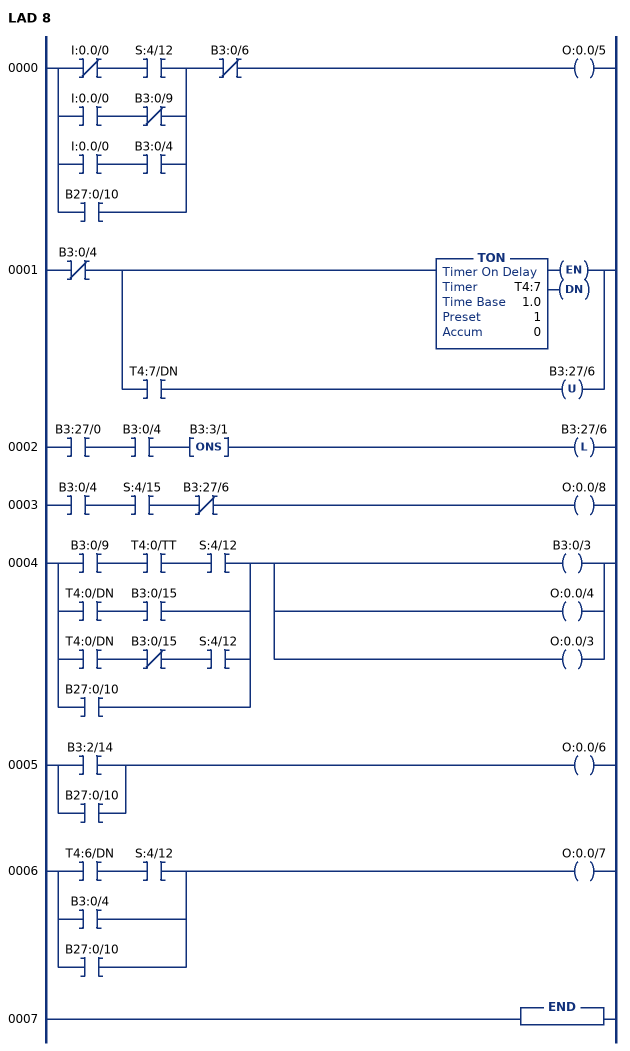
% Rung: 0 %
SOR BST XIO I:0.0/0 XIC S:4/12 NXB XIC I:0.0/0 XIO B3:0/9 NXB XIC I:0.0/0 XIC B3:0/4 NXB XIC B27:0/10 BND XIO B3:0/6 OTE O:0.0/5 EOR
% Rung: 1 %
SOR XIO B3:0/4 BST TON T4:7 1.0 1 0 NXB XIC T4:7/DN OTU B3:27/6 BND EOR
% Rung: 2 %
SOR XIC B3:27/0 XIC B3:0/4 ONS B3:3/1 OTL B3:27/6 EOR
% Rung: 3 %
SOR XIC B3:0/4 XIC S:4/15 XIO B3:27/6 OTE O:0.0/8 EOR
% Rung: 4 %
SOR BST XIC B3:0/9 XIC T4:0/TT XIC S:4/12 NXB XIC T4:0/DN XIC B3:0/15 NXB XIC T4:0/DN XIO B3:0/15 XIC S:4/12 NXB XIC B27:0/10 BND BST OTE B3:0/3 NXB OTE O:0.0/4 NXB OTE O:0.0/3 BND EOR
% Rung: 5 %
SOR BST XIC B3:2/14 NXB XIC B27:0/10 BND OTE O:0.0/6 EOR
% Rung: 6 %
SOR BST XIC T4:6/DN XIC S:4/12 NXB XIC B3:0/4 NXB XIC B27:0/10 BND OTE O:0.0/7 EOR
% Rung: 7 %
SOR END EOR

LADDER 9
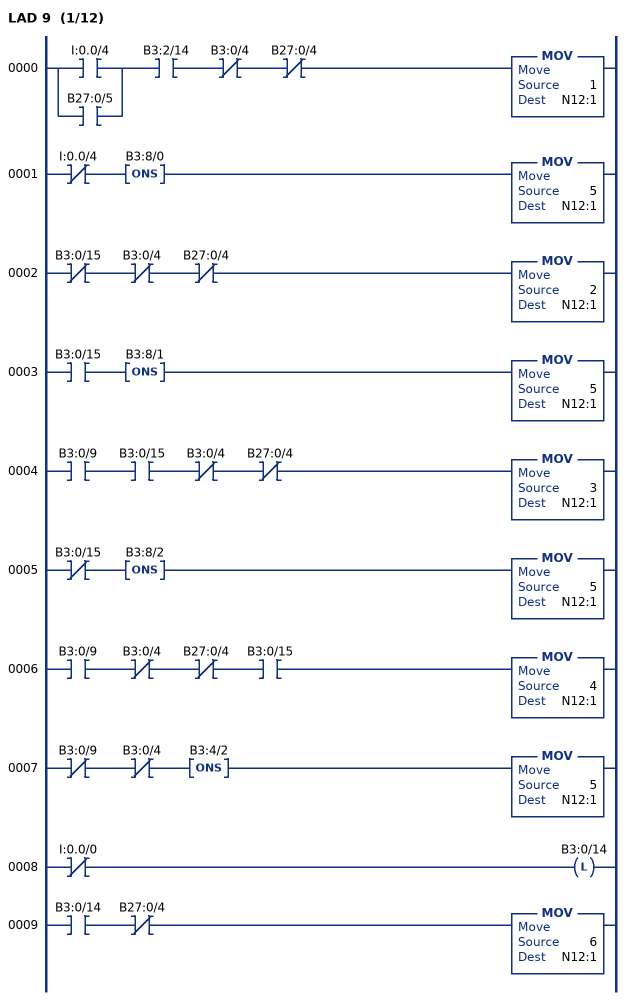
% Rung: 0 %
SOR BST XIC I:0.0/4 NXB XIC B27:0/5 BND XIC B3:2/14 XIO B3:0/4 XIO B27:0/4 MOV 1 N12:1 EOR
% Rung: 1 %
SOR XIO I:0.0/4 ONS B3:8/0 MOV 5 N12:1 EOR
% Rung: 2 %
SOR XIO B3:0/15 XIO B3:0/4 XIO B27:0/4 MOV 2 N12:1 EOR
% Rung: 3 %
SOR XIC B3:0/15 ONS B3:8/1 MOV 5 N12:1 EOR
% Rung: 4 %
SOR XIC B3:0/9 XIC B3:0/15 XIO B3:0/4 XIO B27:0/4 MOV 3 N12:1 EOR
% Rung: 5 %
SOR XIO B3:0/15 ONS B3:8/2 MOV 5 N12:1 EOR
% Rung: 6 %
SOR XIC B3:0/9 XIO B3:0/4 XIO B27:0/4 XIC B3:0/15 MOV 4 N12:1 EOR
% Rung: 7 %
SOR XIO B3:0/9 XIO B3:0/4 ONS B3:4/2 MOV 5 N12:1 EOR
% Rung: 8 %
SOR XIO I:0.0/0 OTL B3:0/14 EOR
% Rung: 9 %
SOR XIC B3:0/14 XIO B27:0/4 MOV 6 N12:1 EOR

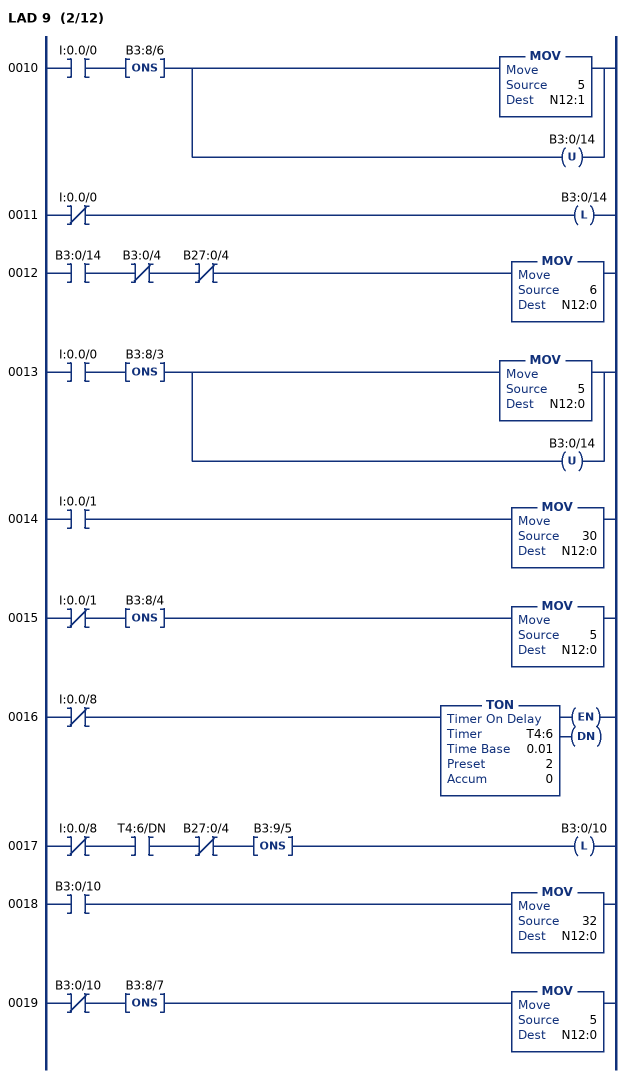
% Rung: 10 %
SOR XIC I:0.0/0 ONS B3:8/6 BST MOV 5 N12:1 NXB OTU B3:0/14 BND EOR
% Rung: 11 %
SOR XIO I:0.0/0 OTL B3:0/14 EOR
% Rung: 12 %
SOR XIC B3:0/14 XIO B3:0/4 XIO B27:0/4 MOV 6 N12:0 EOR
% Rung: 13 %
SOR XIC I:0.0/0 ONS B3:8/3 BST MOV 5 N12:0 NXB OTU B3:0/14 BND EOR
% Rung: 14 %
SOR XIC I:0.0/1 MOV 30 N12:0 EOR
% Rung: 15 %
SOR XIO I:0.0/1 ONS B3:8/4 MOV 5 N12:0 EOR
% Rung: 16 %
SOR XIO I:0.0/8 TON T4:6 0.01 2 0 EOR
% Rung: 17 %
SOR XIO I:0.0/8 XIC T4:6/DN XIO B27:0/4 ONS B3:9/5 OTL B3:0/10 EOR
% Rung: 18 %
SOR XIC B3:0/10 MOV 32 N12:0 EOR
% Rung: 19 %
SOR XIO B3:0/10 ONS B3:8/7 MOV 5 N12:0 EOR

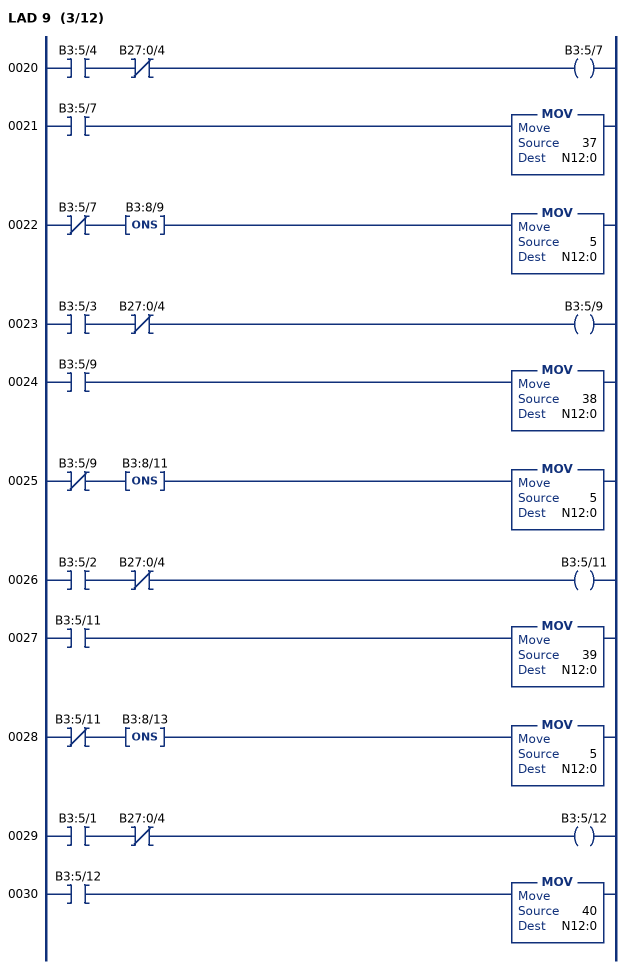
% Rung: 20 %
SOR XIC B3:5/4 XIO B27:0/4 OTE B3:5/7 EOR
% Rung: 21 %
SOR XIC B3:5/7 MOV 37 N12:0 EOR
% Rung: 22 %
SOR XIO B3:5/7 ONS B3:8/9 MOV 5 N12:0 EOR
% Rung: 23 %
SOR XIC B3:5/3 XIO B27:0/4 OTE B3:5/9 EOR
% Rung: 24 %
SOR XIC B3:5/9 MOV 38 N12:0 EOR
% Rung: 25 %
SOR XIO B3:5/9 ONS B3:8/11 MOV 5 N12:0 EOR
% Rung: 26 %
SOR XIC B3:5/2 XIO B27:0/4 OTE B3:5/11 EOR
% Rung: 27 %
SOR XIC B3:5/11 MOV 39 N12:0 EOR
% Rung: 28 %
SOR XIO B3:5/11 ONS B3:8/13 MOV 5 N12:0 EOR
% Rung: 29 %
SOR XIC B3:5/1 XIO B27:0/4 OTE B3:5/12 EOR
% Rung: 30 %
SOR XIC B3:5/12 MOV 40 N12:0 EOR

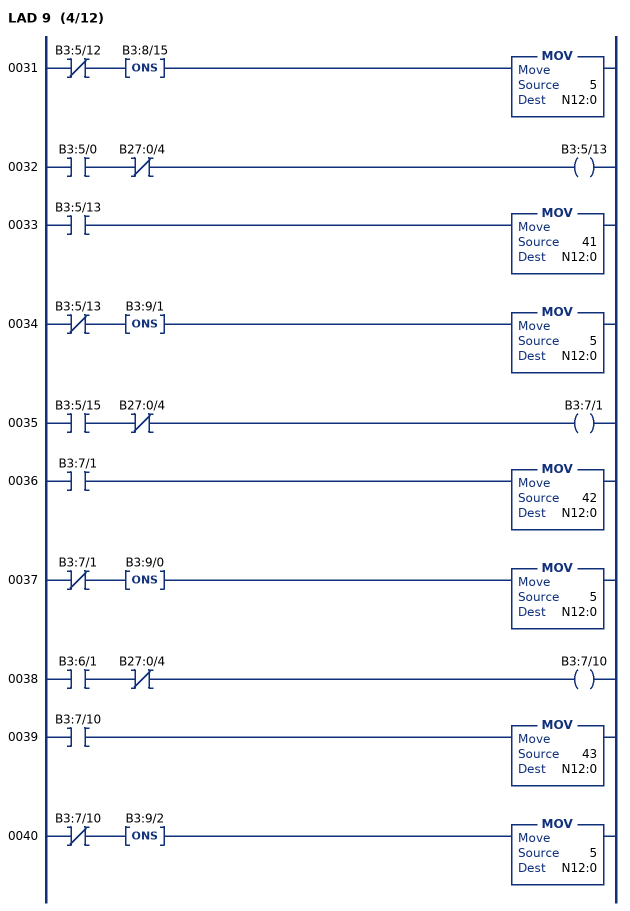
% Rung: 31 %
SOR XIO B3:5/12 ONS B3:8/15 MOV 5 N12:0 EOR
% Rung: 32 %
SOR XIC B3:5/0 XIO B27:0/4 OTE B3:5/13 EOR
% Rung: 33 %
SOR XIC B3:5/13 MOV 41 N12:0 EOR
% Rung: 34 %
SOR XIO B3:5/13 ONS B3:9/1 MOV 5 N12:0 EOR
% Rung: 35 %
SOR XIC B3:5/15 XIO B27:0/4 OTE B3:7/1 EOR
% Rung: 36 %
SOR XIC B3:7/1 MOV 42 N12:0 EOR
% Rung: 37 %
SOR XIO B3:7/1 ONS B3:9/0 MOV 5 N12:0 EOR
% Rung: 38 %
SOR XIC B3:6/1 XIO B27:0/4 OTE B3:7/10 EOR
% Rung: 39 %
SOR XIC B3:7/10 MOV 43 N12:0 EOR
% Rung: 40 %
SOR XIO B3:7/10 ONS B3:9/2 MOV 5 N12:0 EOR

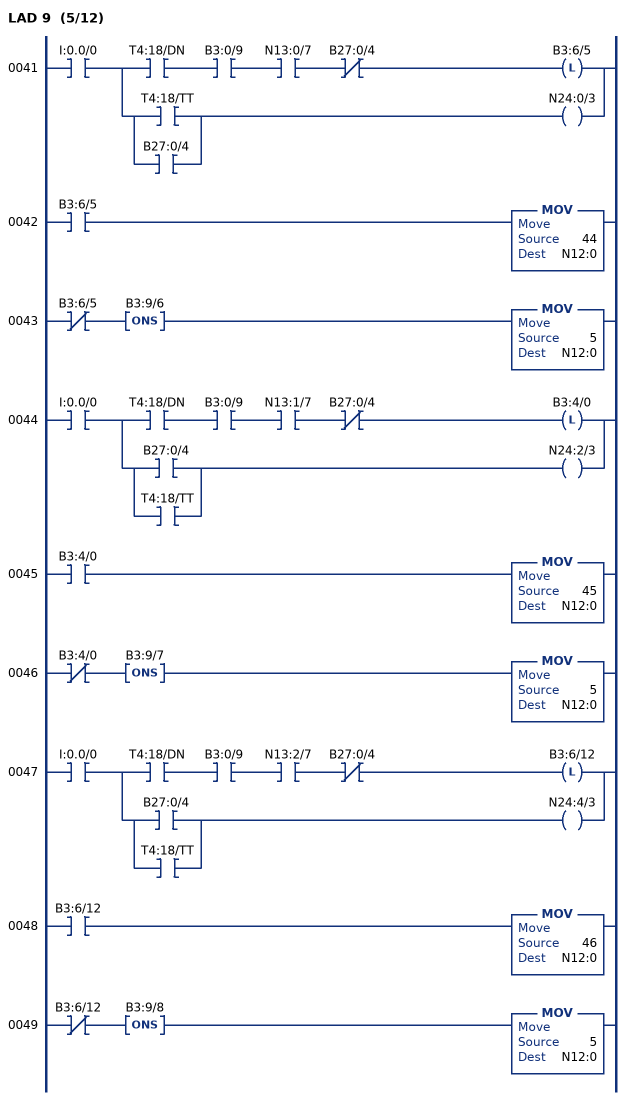
% Rung: 41 %
SOR XIC I:0.0/0 BST XIC T4:18/DN XIC B3:0/9 XIC N13:0/7 XIO B27:0/4 OTL B3:6/5 NXB BST XIC T4:18/TT NXB XIC B27:0/4 BND OTE N24:0/3 BND EOR
% Rung: 42 %
SOR XIC B3:6/5 MOV 44 N12:0 EOR
% Rung: 43 %
SOR XIO B3:6/5 ONS B3:9/6 MOV 5 N12:0 EOR
% Rung: 44 %
SOR XIC I:0.0/0 BST XIC T4:18/DN XIC B3:0/9 XIC N13:1/7 XIO B27:0/4 OTL B3:4/0 NXB BST XIC B27:0/4 NXB XIC T4:18/TT BND OTE N24:2/3 BND EOR
% Rung: 45 %
SOR XIC B3:4/0 MOV 45 N12:0 EOR
% Rung: 46 %
SOR XIO B3:4/0 ONS B3:9/7 MOV 5 N12:0 EOR
% Rung: 47 %
SOR XIC I:0.0/0 BST XIC T4:18/DN XIC B3:0/9 XIC N13:2/7 XIO B27:0/4 OTL B3:6/12 NXB BST XIC B27:0/4 NXB XIC T4:18/TT BND OTE N24:4/3 BND EOR
% Rung: 48 %
SOR XIC B3:6/12 MOV 46 N12:0 EOR
% Rung: 49 %
SOR XIO B3:6/12 ONS B3:9/8 MOV 5 N12:0 EOR

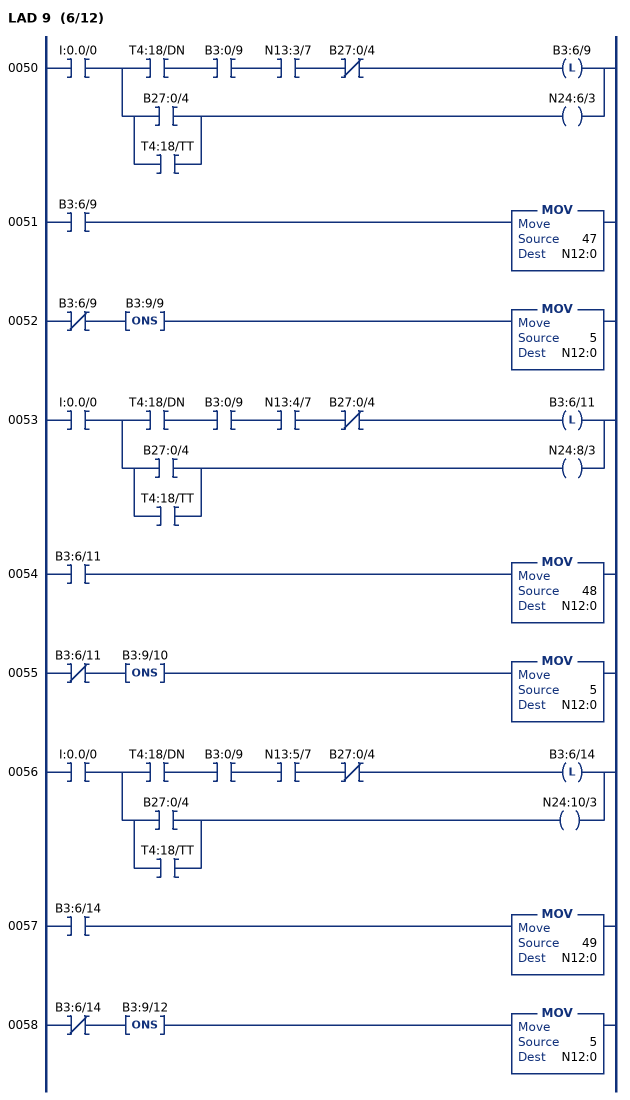
% Rung: 50 %
SOR XIC I:0.0/0 BST XIC T4:18/DN XIC B3:0/9 XIC N13:3/7 XIO B27:0/4 OTL B3:6/9 NXB BST XIC B27:0/4 NXB XIC T4:18/TT BND OTE N24:6/3 BND EOR
% Rung: 51 %
SOR XIC B3:6/9 MOV 47 N12:0 EOR
% Rung: 52 %
SOR XIO B3:6/9 ONS B3:9/9 MOV 5 N12:0 EOR
% Rung: 53 %
SOR XIC I:0.0/0 BST XIC T4:18/DN XIC B3:0/9 XIC N13:4/7 XIO B27:0/4 OTL B3:6/11 NXB BST XIC B27:0/4 NXB XIC T4:18/TT BND OTE N24:8/3 BND EOR
% Rung: 54 %
SOR XIC B3:6/11 MOV 48 N12:0 EOR
% Rung: 55 %
SOR XIO B3:6/11 ONS B3:9/10 MOV 5 N12:0 EOR
% Rung: 56 %
SOR XIC I:0.0/0 BST XIC T4:18/DN XIC B3:0/9 XIC N13:5/7 XIO B27:0/4 OTL B3:6/14 NXB BST XIC B27:0/4 NXB XIC T4:18/TT BND OTE N24:10/3 BND EOR
% Rung: 57 %
SOR XIC B3:6/14 MOV 49 N12:0 EOR
% Rung: 58 %
SOR XIO B3:6/14 ONS B3:9/12 MOV 5 N12:0 EOR

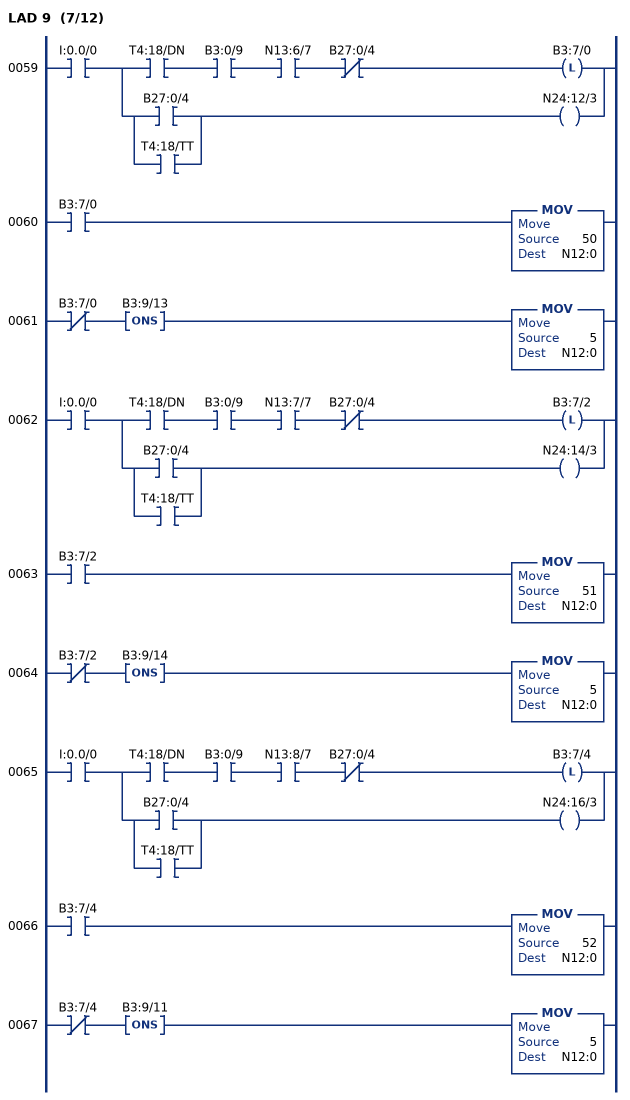
% Rung: 59 %
SOR XIC I:0.0/0 BST XIC T4:18/DN XIC B3:0/9 XIC N13:6/7 XIO B27:0/4 OTL B3:7/0 NXB BST XIC B27:0/4 NXB XIC T4:18/TT BND OTE N24:12/3 BND EOR
% Rung: 60 %
SOR XIC B3:7/0 MOV 50 N12:0 EOR
% Rung: 61 %
SOR XIO B3:7/0 ONS B3:9/13 MOV 5 N12:0 EOR
% Rung: 62 %
SOR XIC I:0.0/0 BST XIC T4:18/DN XIC B3:0/9 XIC N13:7/7 XIO B27:0/4 OTL B3:7/2 NXB BST XIC B27:0/4 NXB XIC T4:18/TT BND OTE N24:14/3 BND EOR
% Rung: 63 %
SOR XIC B3:7/2 MOV 51 N12:0 EOR
% Rung: 64 %
SOR XIO B3:7/2 ONS B3:9/14 MOV 5 N12:0 EOR
% Rung: 65 %
SOR XIC I:0.0/0 BST XIC T4:18/DN XIC B3:0/9 XIC N13:8/7 XIO B27:0/4 OTL B3:7/4 NXB BST XIC B27:0/4 NXB XIC T4:18/TT BND OTE N24:16/3 BND EOR
% Rung: 66 %
SOR XIC B3:7/4 MOV 52 N12:0 EOR
% Rung: 67 %
SOR XIO B3:7/4 ONS B3:9/11 MOV 5 N12:0 EOR

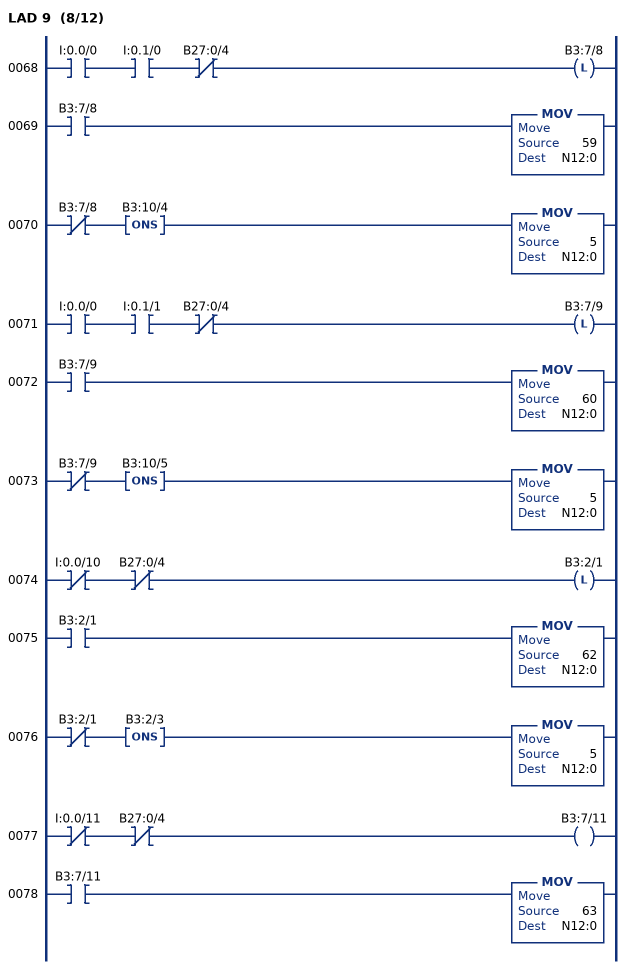
% Rung: 68 %
SOR XIC I:0.0/0 XIC I:0.1/0 XIO B27:0/4 OTL B3:7/8 EOR
% Rung: 69 %
SOR XIC B3:7/8 MOV 59 N12:0 EOR
% Rung: 70 %
SOR XIO B3:7/8 ONS B3:10/4 MOV 5 N12:0 EOR
% Rung: 71 %
SOR XIC I:0.0/0 XIC I:0.1/1 XIO B27:0/4 OTL B3:7/9 EOR
% Rung: 72 %
SOR XIC B3:7/9 MOV 60 N12:0 EOR
% Rung: 73 %
SOR XIO B3:7/9 ONS B3:10/5 MOV 5 N12:0 EOR
% Rung: 74 %
SOR XIO I:0.0/10 XIO B27:0/4 OTL B3:2/1 EOR
% Rung: 75 %
SOR XIC B3:2/1 MOV 62 N12:0 EOR
% Rung: 76 %
SOR XIO B3:2/1 ONS B3:2/3 MOV 5 N12:0 EOR
% Rung: 77 %
SOR XIO I:0.0/11 XIO B27:0/4 OTE B3:7/11 EOR
% Rung: 78 %
SOR XIC B3:7/11 MOV 63 N12:0 EOR

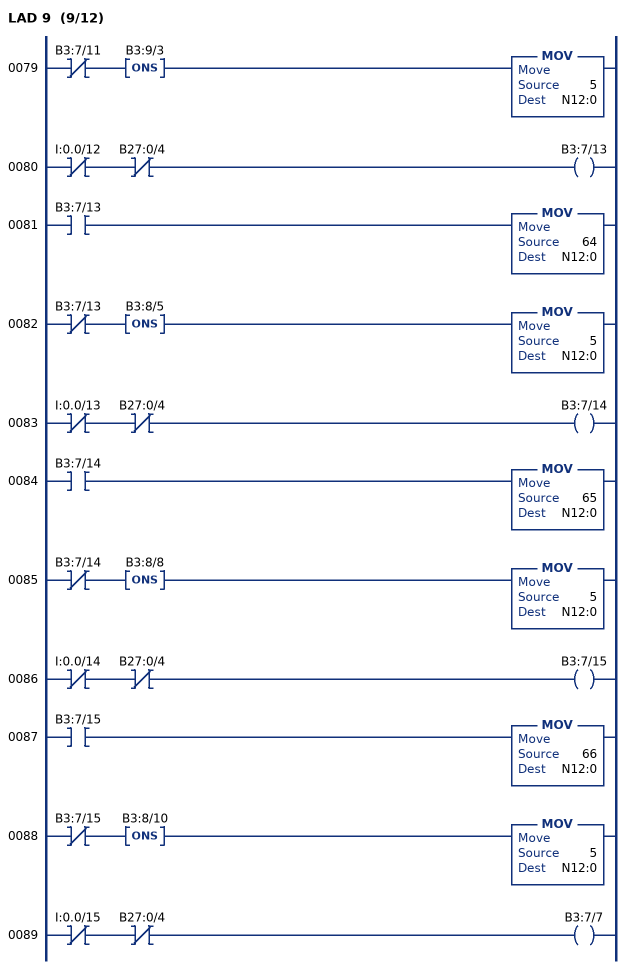
% Rung: 79 %
SOR XIO B3:7/11 ONS B3:9/3 MOV 5 N12:0 EOR
% Rung: 80 %
SOR XIO I:0.0/12 XIO B27:0/4 OTE B3:7/13 EOR
% Rung: 81 %
SOR XIC B3:7/13 MOV 64 N12:0 EOR
% Rung: 82 %
SOR XIO B3:7/13 ONS B3:8/5 MOV 5 N12:0 EOR
% Rung: 83 %
SOR XIO I:0.0/13 XIO B27:0/4 OTE B3:7/14 EOR
% Rung: 84 %
SOR XIC B3:7/14 MOV 65 N12:0 EOR
% Rung: 85 %
SOR XIO B3:7/14 ONS B3:8/8 MOV 5 N12:0 EOR
% Rung: 86 %
SOR XIO I:0.0/14 XIO B27:0/4 OTE B3:7/15 EOR
% Rung: 87 %
SOR XIC B3:7/15 MOV 66 N12:0 EOR
% Rung: 88 %
SOR XIO B3:7/15 ONS B3:8/10 MOV 5 N12:0 EOR
% Rung: 89 %
SOR XIO I:0.0/15 XIO B27:0/4 OTE B3:7/7 EOR

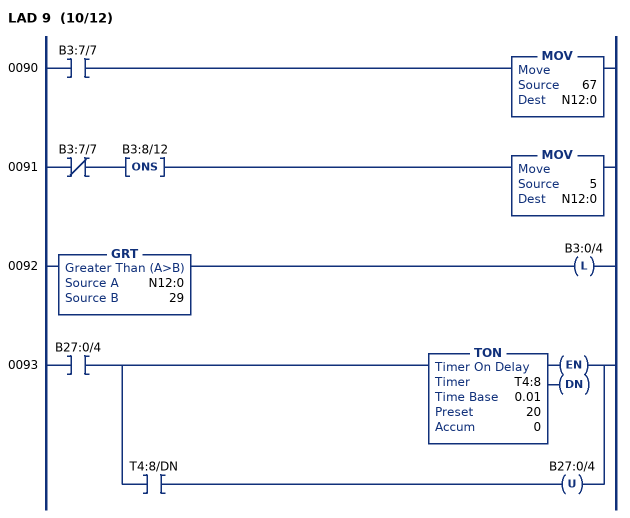
% Rung: 90 %
SOR XIC B3:7/7 MOV 67 N12:0 EOR
% Rung: 91 %
SOR XIO B3:7/7 ONS B3:8/12 MOV 5 N12:0 EOR
% Rung: 92 %
SOR GRT N12:0 29 OTL B3:0/4 EOR
% Rung: 93 %
SOR XIC B27:0/4 BST TON T4:8 0.01 20 0 NXB XIC T4:8/DN OTU B27:0/4 BND EOR

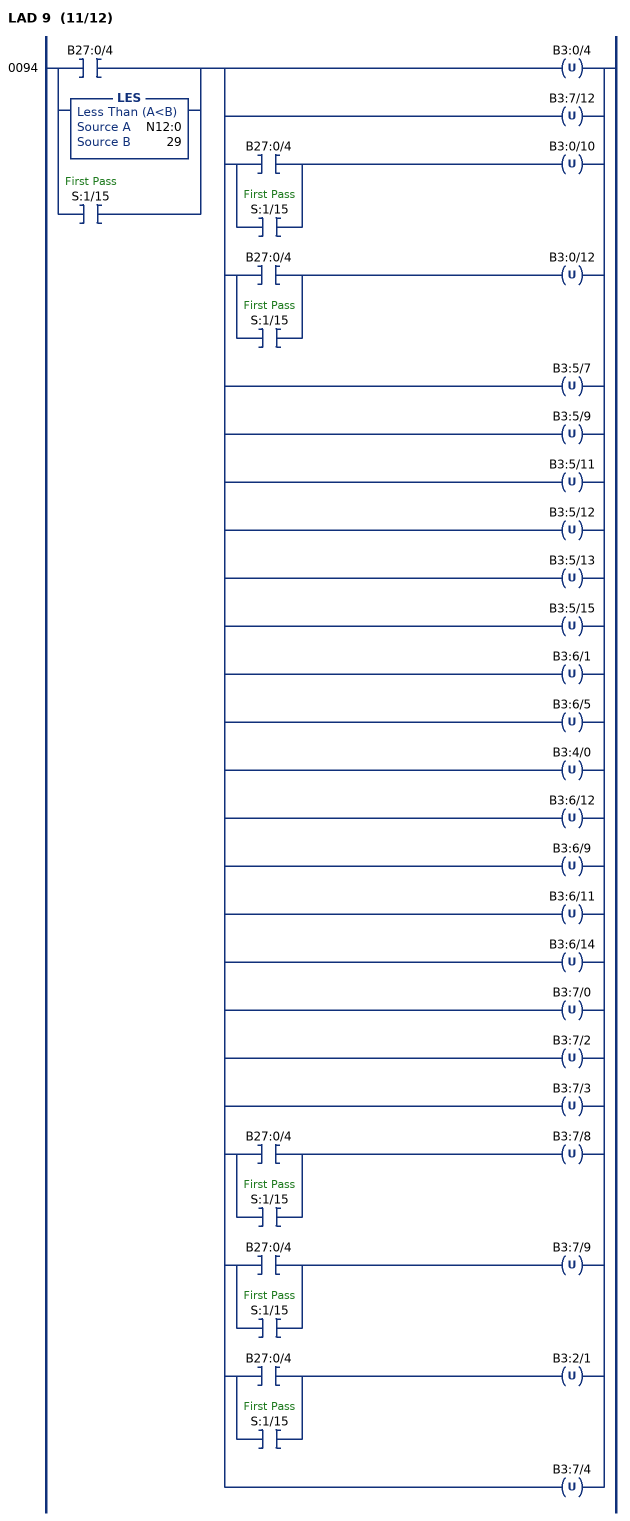
% Rung: 94 %
SOR BST XIC B27:0/4 NXB LES N12:0 29 NXB XIC S:1/15 BND BST OTU B3:0/4 NXB OTU B3:7/12 NXB BST XIC B27:0/4 NXB XIC S:1/15 BND OTU B3:0/10 NXB BST XIC B27:0/4 NXB XIC S:1/15 BND OTU B3:0/12 NXB OTU B3:5/7 NXB OTU B3:5/9 NXB OTU B3:5/11 NXB OTU B3:5/12 NXB OTU B3:5/13 NXB OTU B3:5/15 NXB OTU B3:6/1 NXB OTU B3:6/5 NXB OTU B3:4/0 NXB OTU B3:6/12 NXB OTU B3:6/9 NXB OTU B3:6/11 NXB OTU B3:6/14 NXB OTU B3:7/0 NXB OTU B3:7/2 NXB OTU B3:7/3 NXB BST XIC B27:0/4 NXB XIC S:1/15 BND OTU B3:7/8 NXB BST XIC B27:0/4 NXB XIC S:1/15 BND OTU B3:7/9 NXB BST XIC B27:0/4 NXB XIC S:1/15 BND OTU B3:2/1 NXB OTU B3:7/4 BND EOR
%   S:1/15  "First Pass" %

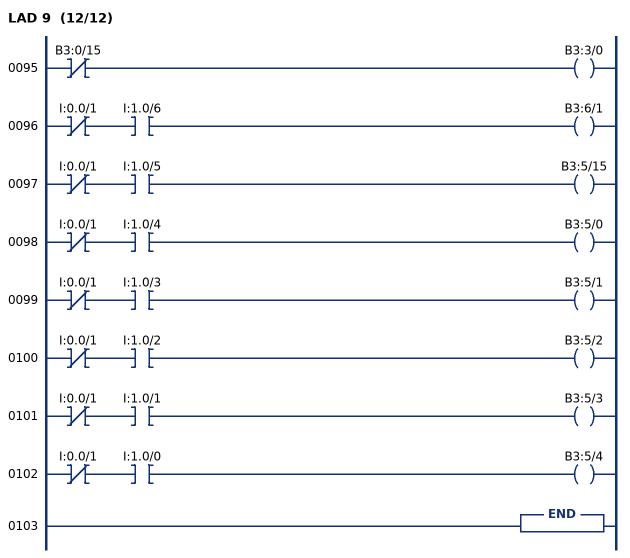
% Rung: 95 %
SOR XIO B3:0/15 OTE B3:3/0 EOR
% Rung: 96 %
SOR XIO I:0.0/1 XIC I:1.0/6 OTE B3:6/1 EOR
% Rung: 97 %
SOR XIO I:0.0/1 XIC I:1.0/5 OTE B3:5/15 EOR
% Rung: 98 %
SOR XIO I:0.0/1 XIC I:1.0/4 OTE B3:5/0 EOR
% Rung: 99 %
SOR XIO I:0.0/1 XIC I:1.0/3 OTE B3:5/1 EOR
% Rung: 100 %
SOR XIO I:0.0/1 XIC I:1.0/2 OTE B3:5/2 EOR
% Rung: 101 %
SOR XIO I:0.0/1 XIC I:1.0/1 OTE B3:5/3 EOR
% Rung: 102 %
SOR XIO I:0.0/1 XIC I:1.0/0 OTE B3:5/4 EOR
% Rung: 103 %
SOR END EOR

LADDER 10
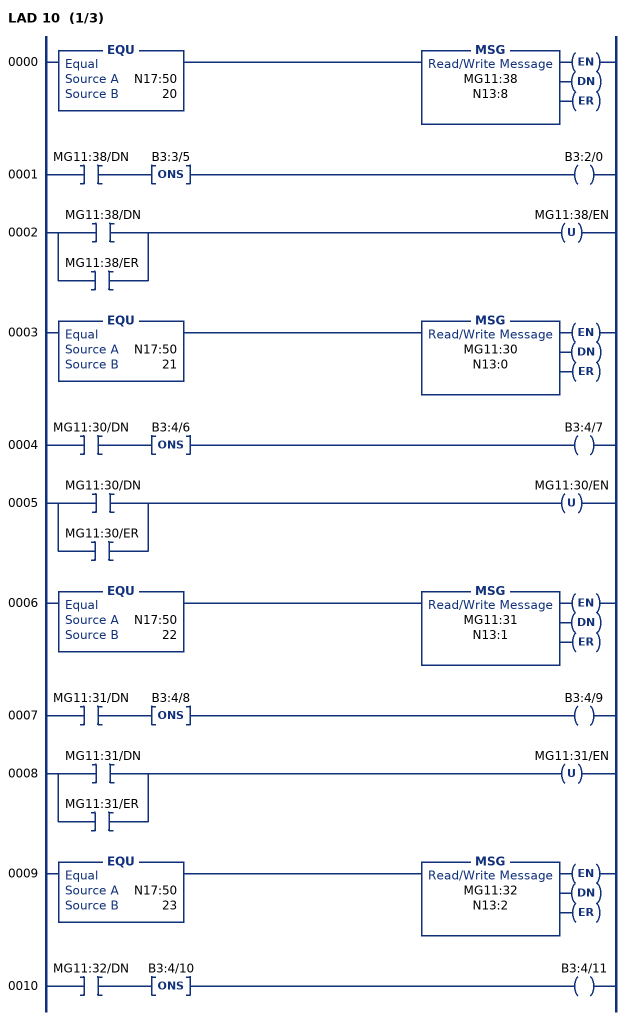
% Rung: 0 %
SOR EQU N17:50 20 MSG MG11:38 N13:8 EOR
%   MSG set-up: 03 Read Holding Registers (4xxxxx) | 5 | 1 | 8449 | N13:8 | 0 | 9 | 0 | CLIENT              :502 | 0 | 0 | ? %
% Rung: 1 %
SOR XIC MG11:38/DN ONS B3:3/5 OTE B3:2/0 EOR
% Rung: 2 %
SOR BST XIC MG11:38/DN NXB XIC MG11:38/ER BND OTU MG11:38/EN EOR
% Rung: 3 %
SOR EQU N17:50 21 MSG MG11:30 N13:0 EOR
%   MSG set-up: 03 Read Holding Registers (4xxxxx) | 5 | 1 | 8449 | N13:0 | 0 | 1 | 0 | CLIENT              :502 | 0 | 0 | ? %
% Rung: 4 %
SOR XIC MG11:30/DN ONS B3:4/6 OTE B3:4/7 EOR
% Rung: 5 %
SOR BST XIC MG11:30/DN NXB XIC MG11:30/ER BND OTU MG11:30/EN EOR
% Rung: 6 %
SOR EQU N17:50 22 MSG MG11:31 N13:1 EOR
%   MSG set-up: 03 Read Holding Registers (4xxxxx) | 5 | 1 | 8449 | N13:1 | 0 | 2 | 0 | CLIENT              :502 | 0 | 0 | ? %
% Rung: 7 %
SOR XIC MG11:31/DN ONS B3:4/8 OTE B3:4/9 EOR
% Rung: 8 %
SOR BST XIC MG11:31/DN NXB XIC MG11:31/ER BND OTU MG11:31/EN EOR
% Rung: 9 %
SOR EQU N17:50 23 MSG MG11:32 N13:2 EOR
%   MSG set-up: 03 Read Holding Registers (4xxxxx) | 5 | 1 | 8449 | N13:2 | 0 | 3 | 0 | CLIENT              :502 | 0 | 0 | ? %
% Rung: 10 %
SOR XIC MG11:32/DN ONS B3:4/10 OTE B3:4/11 EOR

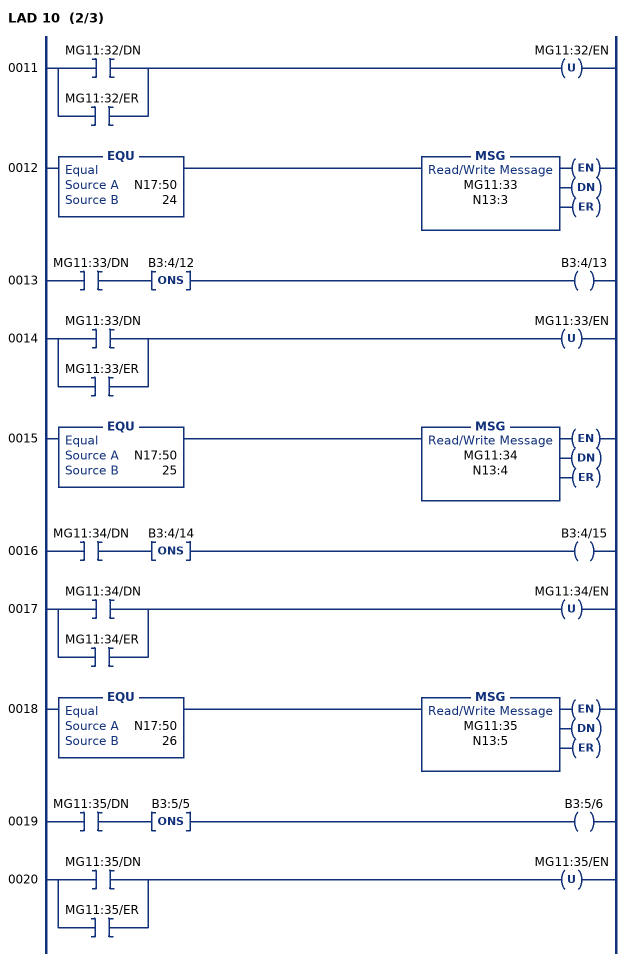
% Rung: 11 %
SOR BST XIC MG11:32/DN NXB XIC MG11:32/ER BND OTU MG11:32/EN EOR
% Rung: 12 %
SOR EQU N17:50 24 MSG MG11:33 N13:3 EOR
%   MSG set-up: 03 Read Holding Registers (4xxxxx) | 5 | 1 | 8449 | N13:3 | 0 | 4 | 0 | CLIENT              :502 | 0 | 0 | ? %
% Rung: 13 %
SOR XIC MG11:33/DN ONS B3:4/12 OTE B3:4/13 EOR
% Rung: 14 %
SOR BST XIC MG11:33/DN NXB XIC MG11:33/ER BND OTU MG11:33/EN EOR
% Rung: 15 %
SOR EQU N17:50 25 MSG MG11:34 N13:4 EOR
%   MSG set-up: 03 Read Holding Registers (4xxxxx) | 5 | 1 | 8449 | N13:4 | 0 | 5 | 0 | CLIENT              :502 | 0 | 0 | ? %
% Rung: 16 %
SOR XIC MG11:34/DN ONS B3:4/14 OTE B3:4/15 EOR
% Rung: 17 %
SOR BST XIC MG11:34/DN NXB XIC MG11:34/ER BND OTU MG11:34/EN EOR
% Rung: 18 %
SOR EQU N17:50 26 MSG MG11:35 N13:5 EOR
%   MSG set-up: 03 Read Holding Registers (4xxxxx) | 5 | 1 | 8449 | N13:5 | 0 | 6 | 0 | CLIENT              :502 | 0 | 0 | ? %
% Rung: 19 %
SOR XIC MG11:35/DN ONS B3:5/5 OTE B3:5/6 EOR
% Rung: 20 %
SOR BST XIC MG11:35/DN NXB XIC MG11:35/ER BND OTU MG11:35/EN EOR

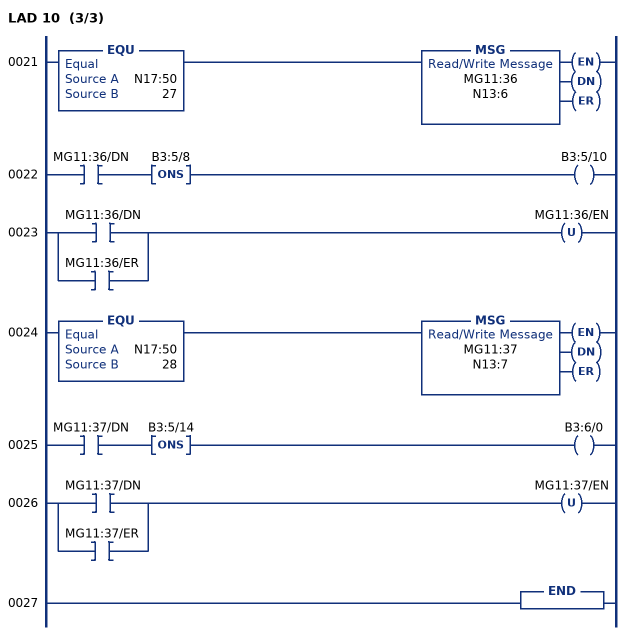
% Rung: 21 %
SOR EQU N17:50 27 MSG MG11:36 N13:6 EOR
%   MSG set-up: 03 Read Holding Registers (4xxxxx) | 5 | 1 | 8449 | N13:6 | 0 | 7 | 0 | CLIENT              :502 | 0 | 0 | ? %
% Rung: 22 %
SOR XIC MG11:36/DN ONS B3:5/8 OTE B3:5/10 EOR
% Rung: 23 %
SOR BST XIC MG11:36/DN NXB XIC MG11:36/ER BND OTU MG11:36/EN EOR
% Rung: 24 %
SOR EQU N17:50 28 MSG MG11:37 N13:7 EOR
%   MSG set-up: 03 Read Holding Registers (4xxxxx) | 5 | 1 | 8449 | N13:7 | 0 | 8 | 0 | CLIENT              :502 | 0 | 0 | ? %
% Rung: 25 %
SOR XIC MG11:37/DN ONS B3:5/14 OTE B3:6/0 EOR
% Rung: 26 %
SOR BST XIC MG11:37/DN NXB XIC MG11:37/ER BND OTU MG11:37/EN EOR
% Rung: 27 %
SOR END EOR

DATA TABLE (non-zero values as saved)
DATA B3
% B3:0 % 0XE890 0X4A96 0X2AAC 0X14A4 0X5540 0XC120 0X0014 0X0062 0XBFB3 0XFFDE
% B3:10 % 0X0033 0X0005 0X8000 0X0007 0X10A8 0X0000 0X0000 0X0000 0X0000 0X0000
DATA T4
% .PRE .ACC %
% T4:0 % 4 0
% T4:1 % 600 600
% T4:2 % 50 50
% T4:3 % 20 20
% T4:4 % 12 0
% T4:5 % 100 0
% T4:6 % 2 0
% T4:7 % 1 0
% T4:8 % 20 0
% T4:9 % 50 50
% T4:10 % 100 0
% T4:11 % 100 100
% T4:12 % 100 100
% T4:13 % 100 100
% T4:14 % 5 5
% T4:15 % 50 0
% T4:16 % 500 500
% T4:17 % 25 0
% T4:18 % 5 0
% T4:19 % 100 0
% T4:20 % 100 0
% T4:21 % 10 0
% T4:24 % 50 0
% T4:25 % 2 0
% T4:29 % 2 0
% T4:36 % 2 2
% T4:37 % 30 0
% T4:38 % 100 0
% T4:39 % 3600 1167
DATA C5
% .PRE .ACC %
% C5:0 % 9999 0
DATA N7
% N7:0 % 3 20 12 600 100 350 0 0 0 0
% N7:10 % 20 80 400 345 890 590 390 710 230 210
% N7:20 % 170 150 400 600 0 0 0 0 0 0
% N7:30 % 180 150 250 150 20 12 700 50 0 0
% N7:40 % 230 210 260 160 22 7 450 110 0 0
% N7:50 % 230 210 170 150 20 12 600 100 0 0
% N7:60 % 180 150 250 150 5 300 600 50 0 0
% N7:70 % 0 0 0 0 250 125 800 0 0 0
% N7:80 % 0 0 0 0 5 300 300 0 0 0
% N7:90 % 0 0 0 0 50 300 500 0 0 0
% N7:100 % 0 0 0 0 3 325 500 0 0 0
% N7:110 % 0 0 0 0 0 0 500 0 0 0
% N7:130 % 50 100 50 100 50 100 100 100 100 0
% N7:140 % 5 100 50 100 50 100 100 100 100 0
% N7:150 % 50 100 50 100 50 100 100 100 100 0
% N7:160 % 50 100 50 100 50 100 100 100 100 0
% N7:170 % 50 100 50 100 50 100 100 100 100 0
% N7:180 % 50 100 50 100 50 100 100 100 100 0
% N7:190 % 2 200 50 100 50 100 100 100 100 0
% N7:200 % 50 100 50 100 50 100 100 100 100 0
% N7:210 % 50 100 50 100 50 100 100 100 100 0
% N7:220 % 50 100 50 100 50 100 100 100 100 0
% N7:230 % 50 100 50 100 50 100 100 100 100 0
DATA F8
% F8:0 % 11.36 11.36 11.36 11.36 11.36
% F8:5 % 11.36 11.36 11.36 11.36 11.36
% F8:10 % 11.36 11.36 0 0 0
DATA N9
% N9:0 % 1 10 10 1 0 31 61 0 0 0
% N9:10 % 0 0 4 0 216 1 1 0 0 0
% N9:20 % 32767 0 0 14124 2841
DATA N10
% N10:0 % 150 150 250 150 230 230 400 220 160 450
% N10:10 % 340 200 400 200 250 300 450 350 260 150
% N10:20 % 160 160 160 160 230 230 400 220 160 500
% N10:30 % 150 150 800 150 230 230 400 220 160 450
% N10:40 % 350 500 550 320 430 450 620 800 210 270
% N10:50 % 200 220 250 200 350 400 550 800 160 0
% N10:60 % 350 500 400 280 420 500 550 800 150 0
% N10:70 % 150 500 550 280 400 400 550 800 250 0
% N10:80 % 250 540 220 260 300 250 300 450 150 0
% N10:90 % 250 250 290 390 400 200 250 200 0 0
% N10:100 % 150 150 350 390 400 200 250 200 0 0
% N10:200 % 1600 3670 2262 870 2770 1364 1060 6200 6131 2680
% N10:210 % 15520 10213 1275 7580 3293 430 2545 2009 230 210
% N10:220 % 260 160 1821 1766 1149 895 2120 947 360 2120
% N10:230 % 1416 360
DATA N12
% N12:0 % 42 6
DATA N13
% N13:0 % 1549 1549 1549 1549 1549 1549 1549 1549 1549 1549
DATA F14
% F14:0 % 0 0 0.4674353 1.505268 0.4674353
% F14:5 % 0.96 0.4674353 0.44991 0.01195719 0.4674353
DATA F15
% F15:0 % 0 3.7 2.5 3.9 2.72
% F15:5 % 3.7 2.75 4.19 4.19 4
% F15:10 % 4 4 4 4 4
% F15:15 % 4 4 4 4 4
% F15:20 % 4
DATA F16
% F16:0 % 25 30 13.5 4 20
% F16:5 % 25 26 54 3.5 5.4
% F16:10 % 25 30 13.5 4 20
% F16:15 % 25 26 54 3.5 5.4
% F16:20 % 20 38 13 3.8 20
% F16:25 % 25 26 53 10 16
% F16:30 % 25 30 13 10 42
% F16:35 % 35 55 1000 5.2 15
% F16:40 % 10 30 4 0.2 12
% F16:45 % 15 15 1400 4 16
% F16:50 % 10 30 7.5 0.3 13
% F16:55 % 18 15 1400 1.2 2.6
% F16:60 % 10 30 7.5 0.3 13
% F16:65 % 18 15 1400 4 9.5
% F16:70 % 10 30 20 1 20
% F16:75 % 20 21 1400 18 17
% F16:80 % 10 30 20 1 20
% F16:85 % 20 21 1400 18 18
% F16:90 % 10 10 1 0.1 16
% F16:95 % 16 16 1400 4 16
% F16:100 % 10 14 3 0 8
% F16:105 % 9.5 4 850 3 19
% F16:110 % 10 30 9 1 19
% F16:115 % 14 19 23 830 19
% F16:120 % 10 30 8 1 19
% F16:125 % 14 19 23 830 19
% F16:130 % 10 10 1 0.1 16
% F16:135 % 16 16 3 1500 16
% F16:140 % 10 35 18 0.1 22
% F16:145 % 17 22 40 825 22
% F16:150 % 10 10 1 0.1 16
% F16:155 % 16 16 3 1500 16
% F16:160 % 10 30 4 1 17
% F16:165 % 11 17 23 830 17
% F16:170 % 10 30 2 1.2 19
% F16:175 % 16 19 20 830 19
% F16:180 % 10 35 18 0.1 22
% F16:185 % 17 22 40 825 22
% F16:190 % 10 10 1 0.1 16
% F16:195 % 16 16 3 1500 16
% F16:200 % 10 10 1 0.1 16
% F16:205 % 16 16 3 1500 16
DATA N17
% N17:0 % 150 200 220 100 165 165 165 50 50 90
% N17:10 % 100 70 70 55 60 60 80 50 60 0
% N17:20 % 100 0 0 0 0 0 0 0 0 0
% N17:50 % 1 0 0 0 0 0 0 0 0 0
DATA F18
% F18:0 % 40 40 194.6793 60.45433 194.6793
% F18:5 % 94.79167 194.6793 202.2627 69.16666 194.6793
DATA N19
% N19:0 % 33 50 690 290 350 900 420 142 350 350
% N19:10 % 350 100 100 100 100
DATA F20
% F20:0 % 0 7 8 7 6
% F20:5 % 7.07 5.428 5.264 6.324 6
% F20:10 % 6 6 6 6 6
% F20:15 % 6 6 6 6 6
% F20:20 % 6
DATA F21
% F21:0 % 0.3030303 0.6 1.452831 0.5037861 0.8284227
% F21:5 % 1.335094 0.4748276 0.853429 1.471631 0.9314801
DATA F22
% F22:0 % 0 0 25.672 7.972 25.672
% F22:5 % 12.5 25.672 26.672 1003.58 25.672
DATA ST23
% ST23:0 % "15.2 OZ ROUND"
% ST23:1 % "13.5 OZ"
% ST23:2 % "15.2 OZ SQUARE"
% ST23:3 % "15.2 OZ ROUND"
% ST23:4 % "#4"
% ST23:5 % "#5"
% ST23:6 % "#6"
% ST23:7 % "#7"
% ST23:8 % "#8"
% ST23:9 % "#9  "
% ST23:10 % "#10  "
% ST23:11 % "#11  future"
% ST23:12 % "#12  future"
% ST23:13 % "#13  future"
% ST23:14 % "#14  future"
% ST23:15 % "#15  future"
% ST23:16 % "#16  future"
% ST23:17 % "#17  future"
% ST23:18 % "#18  future"
% ST23:25 % "#1"
DATA N24
% N24:0 % 17 0 1 0 1 0 1 0 1 0
% N24:10 % 1 0 1 0 1 0 1 0 1 0
% N24:20 % 1 0 0 0 0
DATA ST29
% ST29:0 % "\00\00\00\00\00\00\00\00\00\00\00\00\00\00\00\00\00\00\00\00"
% ST29:1 % "Administrator 4 NEM "
DATA N32
% N32:0 % 18 900 5 5 20 20 4 1 3 0
% N32:10 % 18 900 5 5 20 20 4 2 3 0
% N32:20 % 10 900 5 5 1 1 4 3 3 0
% N32:30 % 10 900 5 5 1 1 4 4 3 0
% N32:40 % 12 900 5 5 1 1 4 5 3 0
% N32:50 % 12 900 5 5 1 1 4 6 3 0
% N32:60 % 12 900 5 5 1 1 4 7 3 0
% N32:70 % 12 900 5 5 1 1 4 8 3 0
% N32:80 % 12 900 5 5 1 1 4 9 3 0
% N32:90 % 10 900 5 5 1 1 4 10 3 0
% N32:100 % 12 900 5 5 1 1 4 11 3 0
% N32:110 % 12 900 5 5 1 1 4 12 3 0
